TYPE Mat32 : ARRAY[1..3, 1..2] OF LREAL; END_TYPE

(* stored: Version 1.1.0.1, ProductVersion 3.1.4024.12
   DUT Mat32: Id {02f043a3-e19a-4b03-8f65-4656fdb2d0e1} *)
